// TIA Portal V20 export
// export: Created 2025-12-01T14:57:27.9326665Z, ExportSetting None, DisplayName Totally Integrated Automation Portal, DisplayVersion V20 Update 3, DisplayName TIA Portal Openness, DisplayVersion V20 Update 3, DisplayName TIA Portal Version Control Interface, DisplayVersion V20 Update 3, DisplayName STEP 7 Professional, DisplayVersion V20 Update 3, DisplayName STEP 7 Safety, DisplayVersion V20 Update 2, DisplayName WinCC Basic/Comfort/Advanced, DisplayVersion V20 Update 3, DisplayName WinCC Professional, DisplayVersion V20 Update 3, DisplayName WinCC Unified, DisplayVersion V20 Update 3
FUNCTION_BLOCK "FB602_EntradaMovil_Lateral_EnCarga_Quimarox"   // FB602, LAD
{ S7_Optimized_Access := 'FALSE' }
// stored: AutoNumber false, SetENOAutomatically false
   VAR_INPUT
      MesaAnterior : UInt;
      MesaDeCarga : UInt;
      ID_Quimarox : UInt;
      ID_Elemento : UInt;
      EnTension : Bool;
      Termico_Tx : Bool;
      Termico_Tilt : Bool;
      pHs_PosicionCarga : Bool;
      pHs_Protrusion : Bool;
      En_PosicionReposo : Bool;
      Corte_PosicionReposo : Bool;
      Corte_PosicionCarga : Bool;
      En_PosicionCarga : Bool;
      PRV_AVTF : Bool;
      PRV_DescargaActiva : Bool;
      V_FILTRO_pHsPresencia : Int;
      Pto_Ajuste_1 : Int;
      Pto_Ajuste_2 : Int;
      Pto_Ajuste_3 : Int;
      Pto_Ajuste_4 : Int;
      Pto_Ajuste_5 : Int;
      Pto_Ajuste_6 : Int;
   END_VAR
   VAR_OUTPUT
      PRV_PTF : Bool;
      PRV_FTF : Bool;
      PararElevador : Bool;
      ElevadorEnLenta : Bool;
      Avance_EntradaMovil : Bool;
      Ir_PosicionReposo : Bool;
      Ir_PosicionCarga : Bool;
   END_VAR
   VAR_IN_OUT
      ROUTING_Destino : UInt;
      ROUTING_Etiqueta : UDInt;
   END_VAR
   VAR
      TMP_EnTension { S7_SetPoint := 'True'} : "FB910_CNT_UHS";
      FILTRO_pHsPresencia { S7_SetPoint := 'True'} : "FB910_CNT_UHS";
      EstadoAsociadoEnMesa : UInt;
      Aux_PeineDeCarga : UInt;
      PresenciaEnReset : Bool;
   END_VAR
   VAR_TEMP
      TMP_PeineDeCarga : UInt;
      TMP_PeineLiberar : UInt;
      MesaQuimarox : UInt;
      VagonReservado : UInt;
      NumeroUT : UInt;
      EsMesaTL : Bool;
      FILTRO_PosicionCarga : Bool;
   END_VAR
BEGIN

NETWORK
TITLE = ERROR - Rearme
/////////////////////////////////////////////////////////////
/////////////////////////////////////////////////////////////
/////////////////////////////////////////////////////////////
// Rearne de Errores
      SET;
      A     "DB902_Estado_ZonaMesa".EstadoMesas[#MesaDeCarga].Rearme_CBx;
      O     "DB902_Estado_ZonaMesa".EstadoMesas[#MesaDeCarga].PerReset_CBx;
      R     "DB900_Estado_Mesas".EstadoVI[#MesaDeCarga].Error_Mx;
      R     "DB900_Estado_Mesas".EstadoVI[#MesaDeCarga].Err_Protusion;
      R     "DB900_Estado_Mesas".EstadoVI[#MesaDeCarga].Err_TOut_Avance_E1_E3;
      R     "DB900_Estado_Mesas".EstadoVI[#MesaDeCarga].Err_Tout_Sacar;
      R     "DB900_Estado_Mesas".EstadoVI[#MesaDeCarga].Err_Tout_Recoger;
      R     "DB900_Estado_Mesas".EstadoVI[#MesaDeCarga].Err_DatosPLC;
      R     "DB900_Estado_Mesas".EstadoVI[#MesaDeCarga].Err_Termico_E1_E3;
      R     "DB900_Estado_Mesas".EstadoVI[#MesaDeCarga].Err_Termico_E2_E4;



NETWORK
TITLE = RECEP OK DE LA ORDEN -- NO SE UTILIZA
/////////////////////////////////////////////////////////////
/////////////////////////////////////////////////////////////
/////////////////////////////////////////////////////////////
// RECEP OK DE LA ORDEN
      SET;
      AN    "DB841_Recepcion".Mesa[#MesaDeCarga].Protocolo.Ord_S00;
      AN    "DB841_Recepcion".Mesa[#MesaDeCarga].Protocolo.Ord_S01;
      AN    "DB841_Recepcion".Mesa[#MesaDeCarga].Protocolo.Ord_S02;
      AN    "DB841_Recepcion".Mesa[#MesaDeCarga].Protocolo.Ord_S03;
      NOT;
      =     "DB840_Emision".Mesa[#MesaDeCarga].Protocolo.RecepOK;



NETWORK
TITLE = HMI - Manual
/////////////////////////////////////////////////////////////
/////////////////////////////////////////////////////////////
/////////////////////////////////////////////////////////////
// Para HMI >>> Manual
      SET;
      O     "DB902_Estado_ZonaMesa".EstadoMesas[#MesaDeCarga].Manual_CBx;
      =     "DB900_Estado_Mesas".EstadoVI[#MesaDeCarga].Manual;



NETWORK
TITLE = HMI - Entradas y Salidas de la Mesa
/////////////////////////////////////////////////////////////
/////////////////////////////////////////////////////////////
/////////////////////////////////////////////////////////////
// Entradas
      SET;
      A     #pHs_PosicionCarga;
      =     "DB900_Estado_Mesas".EstadoVI[#MesaDeCarga].En_PHS_1;
      SET;
      A     #pHs_Protrusion;
      =     "DB900_Estado_Mesas".EstadoVI[#MesaDeCarga].En_pHs_Prot1;

      SET;
      A     #Termico_Tx;
      =     "DB900_Estado_Mesas".EstadoVI[#MesaDeCarga].En_Termico1;
      SET;
      A     #Termico_Tilt;
      =     "DB900_Estado_Mesas".EstadoVI[#MesaDeCarga].En_Termico2;

      SET;
      A     #En_PosicionReposo;
      =     "DB904_Estado_Maquinas".EstadoVI[#MesaDeCarga].Byte8_bit4;
      SET;
      A     #Corte_PosicionReposo;
      =     "DB904_Estado_Maquinas".EstadoVI[#MesaDeCarga].Byte7_bit6;
      SET;
      A     #Corte_PosicionCarga;
      =     "DB904_Estado_Maquinas".EstadoVI[#MesaDeCarga].Byte7_bit7;
      SET;
      A     #En_PosicionCarga;
      =     "DB904_Estado_Maquinas".EstadoVI[#MesaDeCarga].Byte8_bit5;


// Salidas
      SET;
      A     #Avance_EntradaMovil;
      =     "DB900_Estado_Mesas".EstadoVI[#MesaDeCarga].Sa_Rod_Avance;
      SET;
      A     #Ir_PosicionReposo;
      =     "DB900_Estado_Mesas".EstadoVI[#MesaDeCarga].Sa_Trans_Baj;
      SET;
      A     #Ir_PosicionCarga;
      =     "DB900_Estado_Mesas".EstadoVI[#MesaDeCarga].Sa_Trans_Sub;



NETWORK
TITLE = Comprobacion de que la MESA es de TRACKING
/////////////////////////////////////////////////////////////
/////////////////////////////////////////////////////////////
/////////////////////////////////////////////////////////////
// Comprobar si es una Mesa de Tracking o Routing
      SET;
      A     "DB850_DefinicionMesas".Mesa[#MesaDeCarga].ConfigMesa.MesaTL;
      =     #EsMesaTL;



REGION Network 6: TMP - Espera En Tension
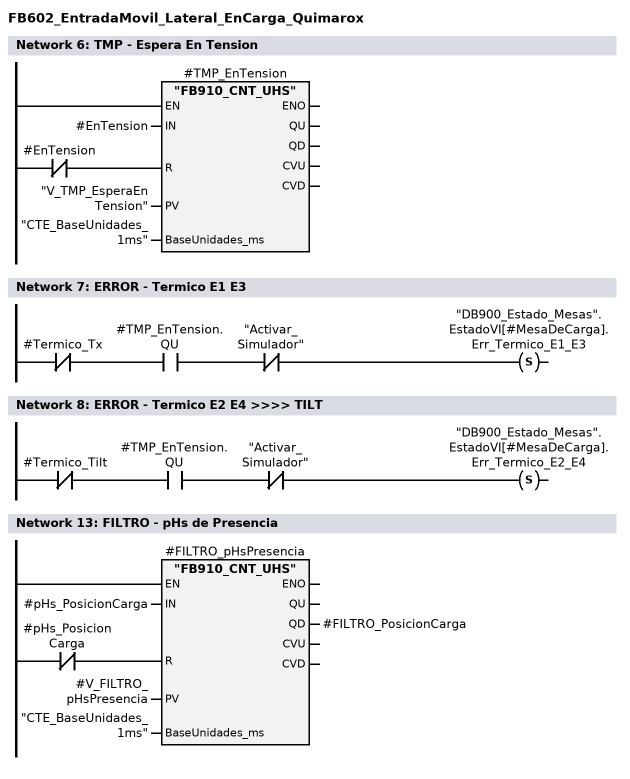
   RUNG wire#powerrail
      #TMP_EnTension(R := wire#w1, IN := #EnTension, PV := "V_TMP_EsperaEnTension", BaseUnidades_ms := "CTE_BaseUnidades_1ms", QU =>, QD =>, CVU =>, CVD =>)
   END_RUNG
   RUNG wire#powerrail
      I_Contact( #EnTension )
   END_RUNG wire#w1
   // the same network as SCL:
   #TMP_EnTension(IN := #EnTension,   // "FB910_CNT_UHS"
                  R := NOT #EnTension,
                  PV := "V_TMP_EsperaEnTension",
                  BaseUnidades_ms := "CTE_BaseUnidades_1ms");
END_REGION

REGION Network 7: ERROR - Termico E1 E3
   RUNG wire#powerrail
      I_Contact( #Termico_Tx )
      Contact( #TMP_EnTension.QU )
      I_Contact( "Activar_Simulador" )
      S_Coil( "DB900_Estado_Mesas".EstadoVI[#MesaDeCarga].Err_Termico_E1_E3 )
   END_RUNG
   // the same network as SCL:
   IF NOT #Termico_Tx AND #TMP_EnTension.QU AND NOT "Activar_Simulador" THEN
       "DB900_Estado_Mesas".EstadoVI[#MesaDeCarga].Err_Termico_E1_E3 := TRUE;
   END_IF;
END_REGION

REGION Network 8: ERROR - Termico E2 E4 >>>> TILT
   RUNG wire#powerrail
      I_Contact( #Termico_Tilt )
      Contact( #TMP_EnTension.QU )
      I_Contact( "Activar_Simulador" )
      S_Coil( "DB900_Estado_Mesas".EstadoVI[#MesaDeCarga].Err_Termico_E2_E4 )
   END_RUNG
   // the same network as SCL:
   IF NOT #Termico_Tilt AND #TMP_EnTension.QU AND NOT "Activar_Simulador" THEN
       "DB900_Estado_Mesas".EstadoVI[#MesaDeCarga].Err_Termico_E2_E4 := TRUE;
   END_IF;
END_REGION

NETWORK
TITLE = INICIALIZACION Previa
/////////////////////////////////////////////////////////////
/////////////////////////////////////////////////////////////
/////////////////////////////////////////////////////////////
      CLR;
      =     #PRV_PTF;
      =     #PRV_FTF;
      CLR;
      =     #ElevadorEnLenta;
      =     #PararElevador;
      =     #Avance_EntradaMovil;
      =     #Ir_PosicionReposo;
      =     #Ir_PosicionCarga;

      CLR;
      =     "DB900_Estado_Mesas".EstadoVI[#MesaDeCarga].Etapas_Reset;
      =     "DB900_Estado_Mesas".EstadoVI[#MesaDeCarga].Etapa_Vacia;
      =     "DB900_Estado_Mesas".EstadoVI[#MesaDeCarga].Etapa_Cargada;
      =     "DB900_Estado_Mesas".EstadoVI[#MesaDeCarga].Etapas_Carga_E1;
      =     "DB900_Estado_Mesas".EstadoVI[#MesaDeCarga].Etapas_Descarga_S0;



NETWORK
TITLE = SISTEMA - Paro Blando
/////////////////////////////////////////////////////////////
/////////////////////////////////////////////////////////////
/////////////////////////////////////////////////////////////
// - Inicializar Variables de PARO BLANDO
      CLR;
      =     "DB900_Estado_Mesas".EstadoVI[#MesaDeCarga].Paro_Blando;

/////////////////////////////////////////////////////////////
// - Existe PARO BLANDO ???
      SET;
      AN    "DB902_Estado_ZonaMesa".EstadoMesas[#MesaDeCarga].ParoBlando_CBx;
      JC    NoRealizandose_ParoBlando;

/////////////////////////////////////////////////////////////
// - Fin de PARO BLANDO
      SET;
      =     "DB900_Estado_Mesas".EstadoVI[#MesaDeCarga].Paro_Blando;


/////////////////////////////////////////////////////////////
/////////////////////////////////////////////////////////////
/////////////////////////////////////////////////////////////
// - Final Tratamiento del PARO BLANDO
NoRealizandose_ParoBlando:NOP   0;



NETWORK
TITLE = SISTEMA - Reset
/////////////////////////////////////////////////////////////
/////////////////////////////////////////////////////////////
/////////////////////////////////////////////////////////////
// -- Inicializar Variables de RESET
      SET;
      AN    "DB902_Estado_ZonaMesa".EstadoMesas[#MesaDeCarga].PerReset_CBx;
      R     "DB900_Estado_Mesas".EstadoVI[#MesaDeCarga].Fin_VI;
      R     #PresenciaEnReset;

/////////////////////////////////////////////////////////////
/////////////////////////////////////////////////////////////
/////////////////////////////////////////////////////////////
// - Existe RESET ??
      SET;
      AN    "DB902_Estado_ZonaMesa".EstadoMesas[#MesaDeCarga].PerReset_CBx;
      JC    NoRealizandose_Reset;

      L     0;  // Estado de La Mesa = 0
      T     #EstadoAsociadoEnMesa;
      SET;
      =     "DB900_Estado_Mesas".EstadoVI[#MesaDeCarga].Etapas_Reset;

/////////////////////////////////////////////////////////////
/////////////////////////////////////////////////////////////
/////////////////////////////////////////////////////////////
// - Emision de Presencia en caso de Reset
      SET;  // Presencia >>> Reset Total
      A     #FILTRO_PosicionCarga;
      AN    #PresenciaEnReset;
      A     "DB831_Mesas".Mesas[#MesaDeCarga].Memorias.M_ResetTotal;
      JC    Enviar_PresenciaEnResetTotal;

      SET;  // Presencia >>> Reset Parcial
      A     #FILTRO_PosicionCarga;
      A     "DB831_Mesas".Mesas[#MesaDeCarga].Memorias.M_ResetParcial;
      AN    #PresenciaEnReset;
      JC    Enviar_PresenciaEnResetParcial;

      JU    Final_PresenciaEnReset;

// - Presencia en Reset TOTAL >>> Enviar NUUT
Enviar_PresenciaEnResetTotal:NOP   0;
      CALL  "FC723_InsertarUT_EnMesa"
      ( MesaActual := #MesaDeCarga,
        NumeroUT   := #NumeroUT
      );
      L     132;  // Envio de Nueva UT en RESET
      T     "DB812_UTs_Control".UT[#NumeroUT].EstadoEventoAGenerar;

      SET;  // Ya esta Avisado el JdT
      S     #PresenciaEnReset;

      JU    Final_PresenciaEnReset;

// - Presencia en Reset Parcial >>> Enviar LOCA en Reset Pantalla
Enviar_PresenciaEnResetParcial:NOP   0;
      L     "DB810_ColasMesas".Colas[#MesaDeCarga].UT_PrimeraMesa;
      T     #NumeroUT;

      L     #NumeroUT;  // Comprobar que Existe UT
      L     0;
      ==I;
      JC    ErrorDatosCargada;

      L     101;  // Envio de LOCA en RESET
      T     "DB812_UTs_Control".UT[#NumeroUT].EstadoEventoAGenerar;

      SET;  // Ya esta Avisado el JdT
      S     #PresenciaEnReset;

      JU    Final_PresenciaEnReset;

// - Final de la Presencia En Reset
Final_PresenciaEnReset:NOP   0;


/////////////////////////////////////////////////////////////
/////////////////////////////////////////////////////////////
/////////////////////////////////////////////////////////////
// - Fin de RESET
      SET;  // Con Presencia de Carga >>> TOTAL
      A(;
      L     "DB810_ColasMesas".Colas[#MesaDeCarga].UT_PrimeraMesa;
      L     0;
      ==I;
      );
      A     #FILTRO_PosicionCarga;
      A     #PresenciaEnReset;
      A     "DB831_Mesas".Mesas[#MesaDeCarga].Memorias.M_ResetTotal;
      S     "DB900_Estado_Mesas".EstadoVI[#MesaDeCarga].Fin_VI;

      SET;  // Con Presencia de Carga >>> PARCIAL
      A     #FILTRO_PosicionCarga;
      A     #PresenciaEnReset;
      A     "DB831_Mesas".Mesas[#MesaDeCarga].Memorias.M_ResetParcial;
      S     "DB900_Estado_Mesas".EstadoVI[#MesaDeCarga].Fin_VI;

      SET;  // Sin Presencia de Carga
      AN    #FILTRO_PosicionCarga;
      S     "DB900_Estado_Mesas".EstadoVI[#MesaDeCarga].Fin_VI;

      BE;

/////////////////////////////////////////////////////////////
/////////////////////////////////////////////////////////////
/////////////////////////////////////////////////////////////
// - Final Tratamiento del RESET
NoRealizandose_Reset:NOP   0;



NETWORK
TITLE = >>>>>>>>>>>>>>>>>>>>>>>>>>>>>>>>>>>>>>>>>>>>>>>>>>>>>>>>>>>>>>>>>>>

REGION Network 13: FILTRO - pHs de Presencia
   RUNG wire#powerrail
      #FILTRO_pHsPresencia(R := wire#w1, IN := #pHs_PosicionCarga, PV := #V_FILTRO_pHsPresencia, BaseUnidades_ms := "CTE_BaseUnidades_1ms", QU =>, QD => #FILTRO_PosicionCarga, CVU =>, CVD =>)
   END_RUNG
   RUNG wire#powerrail
      I_Contact( #pHs_PosicionCarga )
   END_RUNG wire#w1
   // the same network as SCL:
   #FILTRO_pHsPresencia(IN := #pHs_PosicionCarga,   // "FB910_CNT_UHS"
                        R := NOT #pHs_PosicionCarga,
                        PV := #V_FILTRO_pHsPresencia,
                        BaseUnidades_ms := "CTE_BaseUnidades_1ms",
                        QD => #FILTRO_PosicionCarga);
END_REGION

NETWORK
TITLE = >>>>>>>>>>>>>>>>>>>>>>>>>>>>>>>>>>>>>>>>>>>>>>>>>>>>>>>>>>>>>>>>>>>

NETWORK
TITLE = Disrtibucion >>> Control Etapa Activa
/////////////////////////////////////////////////////////////////////////////////////
/////////////////////////////////////////////////////////////////////////////////////
/////////////////////////////////////////////////////////////////////////////////////
// listado de saltos de programa
      L     #EstadoAsociadoEnMesa;
      JL    ESTADO_PorDefecto;

      JU    ETAPA_00_EnReset;
      JU    ETAPA_01_EnReposo;

      JU    ETAPA_02_PrevioCarga_ComprobarRuta;
      JU    ETAPA_03_PrevioCarga_ReservaPeine;
      JU    ETAPA_04_PrevioCarga_Sincroniza;
      JU    ETAPA_05_PrevioCarga_MoverPosicionDeCarga;

      JU    ETAPA_06_Cargando;
      JU    ETAPA_07_FinDeCarga;
      JU    ETAPA_08_CargaDelPeine;
      JU    ETAPA_09_MoverPosicionReposo;

// --- CARGADO
      JU    ETAPA_10_Reset_MoverPosicionDeReposo;
      JU    ETAPA_11_Reset_ComprobarRuta;
      JU    ETAPA_12_Reset_ReservaPeine;
      JU    ETAPA_13_Reset_Sincroniza;
      JU    ETAPA_14_Reset_MoverPosicionDeCarga;

// --- VACIO
      JU    ETAPA_15_Reset_MoverPosicionDeReposo;

ESTADO_PorDefecto:JU    FinFuncion;







NETWORK
TITLE = ETAPA 00 >>> Etapa Reset
/////////////////////////////////////////////////////////////////////////////////////
/////////////////////////////////////////////////////////////////////////////////////
/////////////////////////////////////////////////////////////////////////////////////
ETAPA_00_EnReset:NOP   0;
      SET;
      =     "DB900_Estado_Mesas".EstadoVI[#MesaDeCarga].Etapas_Reset;


/////////////////////////////////////////////////////////////////////////////////////
// error de protusion
      SET;
      AN    #pHs_Protrusion;
      JC    ErrorProtrusion;

/////////////////////////////////////////////////////////////////////////////////////
// Tiene que estar en Marcha y Sin Error para continuar
      SET;
      AN    "DB902_Estado_ZonaMesa".EstadoMesas[#MesaDeCarga].Marcha_CBx;
      O     "DB902_Estado_ZonaMesa".EstadoMesas[#MesaDeCarga].Error_CBx;
      JC    ET00_PararElevador;


/////////////////////////////////////////////////////////////////////////////////////
/////////////////////////////////////////////////////////////////////////////////////
//  Vacio >>> No esta en Reposo
      SET;
      AN    #FILTRO_PosicionCarga;
      AN    #En_PosicionReposo;
      JC    ET00_IrEtapa_15_MoverPosicionReposo;

//  Vacio >>> Esta en Reposo
      SET;
      AN    #FILTRO_PosicionCarga;
      A     #En_PosicionReposo;
      JC    ET00_IrEtapa_01_EnReposo;


/////////////////////////////////////////////////////////////////////////////////////
/////////////////////////////////////////////////////////////////////////////////////
//  Lleno >>> No Esta en Reposo
      SET;
      A     #FILTRO_PosicionCarga;
      AN    #En_PosicionReposo;
      JC    ET00_IrEtapa_10_Reset_MoverPosicionDeReposo;

//  Lleno >>> Esta en Reposo
      SET;
      A     #FILTRO_PosicionCarga;
      A     #En_PosicionReposo;
      JC    ET00_IrEtapa_11_Reset_ComprobarRuta;

      BE;


/////////////////////////////////////////////////////////////////////////////////////
/////////////////////////////////////////////////////////////////////////////////////
/////////////////////////////////////////////////////////////////////////////////////
ET00_PararElevador:NOP   0;
      SET;
      =     #PararElevador;
      BE;


/////////////////////////////////////////////////////////////////////////////////////
/////////////////////////////////////////////////////////////////////////////////////
/////////////////////////////////////////////////////////////////////////////////////
ET00_IrEtapa_01_EnReposo:NOP   0;
      L     1;
      T     #EstadoAsociadoEnMesa;
      JU    ETAPA_01_EnReposo;

/////////////////////////////////////////////////////////////////////////////////////
ET00_IrEtapa_15_MoverPosicionReposo:NOP   0;
      L     15;
      T     #EstadoAsociadoEnMesa;
      JU    ETAPA_15_Reset_MoverPosicionDeReposo;

/////////////////////////////////////////////////////////////////////////////////////
ET00_IrEtapa_11_Reset_ComprobarRuta:NOP   0;
      L     11;
      T     #EstadoAsociadoEnMesa;
      JU    ETAPA_11_Reset_ComprobarRuta;

/////////////////////////////////////////////////////////////////////////////////////
ET00_IrEtapa_10_Reset_MoverPosicionDeReposo:NOP   0;
      L     10;
      T     #EstadoAsociadoEnMesa;
      JU    ETAPA_10_Reset_MoverPosicionDeReposo;




NETWORK
TITLE = ETAPA 01 >>> Etapa Reposo >>> Esta Vacia
/////////////////////////////////////////////////////////////////////////////////////
/////////////////////////////////////////////////////////////////////////////////////
/////////////////////////////////////////////////////////////////////////////////////
// estado reposo
ETAPA_01_EnReposo:NOP   0;
      SET;
      =     "DB900_Estado_Mesas".EstadoVI[#MesaDeCarga].Etapa_Vacia;


/////////////////////////////////////////////////////////////////////////////////////
// error de protusion
      SET;
      AN    #pHs_Protrusion;
      JC    ErrorProtrusion;

/////////////////////////////////////////////////////////////////////////////////////
/////////////////////////////////////////////////////////////////////////////////////
/////////////////////////////////////////////////////////////////////////////////////
// Si Viene un Peine >>> Reservado para el Elemento >>> LIBERAR Peine
      SET;  // --- Sin Ventana
      AN    "DB602_ElementosQuimarox".Quimarox[#ID_Quimarox].Elementos[#ID_Elemento].Hay_Carrier_en_ventana;
      JC    ET01_PorReserva_NoLiberarPeine;

      L     "DB602_ElementosQuimarox".Quimarox[#ID_Quimarox].Elementos[#ID_Elemento].Numero_carrier;
      T     #TMP_PeineLiberar;

      SET;  // --- Sin Reserva
      AN    "DB601_PeinesQuimarox".Quimarox[#ID_Quimarox].vagon[#TMP_PeineLiberar].vagon_reservado_carga;
      JC    ET01_PorReserva_NoLiberarPeine;

      SET;  // --- No es para el elemento
      L     "DB601_PeinesQuimarox".Quimarox[#ID_Quimarox].vagon[#TMP_PeineLiberar].punto_entrada_carga;
      L     #ID_Elemento;
      <>I;
      JC    ET01_PorReserva_NoLiberarPeine;

/////////////////////////////////////////////////////////////////////////////////////
      SET;  // --- Liberar Peine
      R     "DB601_PeinesQuimarox".Quimarox[#ID_Quimarox].vagon[#TMP_PeineLiberar].vagon_reservado_carga;

      L     0;
      T     "DB601_PeinesQuimarox".Quimarox[#ID_Quimarox].vagon[#TMP_PeineLiberar].punto_entrada_carga;

/////////////////////////////////////////////////////////////////////////////////////
ET01_PorReserva_NoLiberarPeine:NOP   0;


/////////////////////////////////////////////////////////////////////////////////////
// Esta poscionado Correctamente
      SET;
      AN    #PRV_AVTF;
      AN    #FILTRO_PosicionCarga;
      A     #pHs_Protrusion;
      AN    #En_PosicionReposo;
      JC    ET01_IrEtapa_09_MoverPosicionReposo;

/////////////////////////////////////////////////////////////////////////////////////
      SET;
      AN    #PRV_AVTF;
      AN    #FILTRO_PosicionCarga;
      A     #pHs_Protrusion;
      JC    FinFuncion;

/////////////////////////////////////////////////////////////////////////////////////
      SET;
      A     #PRV_AVTF;
      AN    #FILTRO_PosicionCarga;
      A     #pHs_Protrusion;
      JC    ET01_IrEtapa_02_PrevioCarga_ComprobarRuta;

      BE;


/////////////////////////////////////////////////////////////////////////////////////
ET01_IrEtapa_09_MoverPosicionReposo:NOP   0;
      L     9;
      T     #EstadoAsociadoEnMesa;
      JU    ETAPA_09_MoverPosicionReposo;

/////////////////////////////////////////////////////////////////////////////////////
ET01_IrEtapa_02_PrevioCarga_ComprobarRuta:NOP   0;
      L     2;  // tengo una caja, paso a extraer orden
      T     #EstadoAsociadoEnMesa;
      JU    ETAPA_02_PrevioCarga_ComprobarRuta;



NETWORK
TITLE = ETAPA 02 >>> Comprobar Ruta
/////////////////////////////////////////////////////////////////////////////////////
/////////////////////////////////////////////////////////////////////////////////////
/////////////////////////////////////////////////////////////////////////////////////
// Extraer Destino
ETAPA_02_PrevioCarga_ComprobarRuta:NOP   0;
      SET;
      =     "DB900_Estado_Mesas".EstadoVI[#MesaDeCarga].Etapa_Vacia;


/////////////////////////////////////////////////////////////////////////////////////
      SET;
      AN    #pHs_Protrusion;
      JC    ErrorProtrusion;

/////////////////////////////////////////////////////////////////////////////////////
/// --- Comprobacion del TIPO de MESA
      SET;
      AN    #EsMesaTL;
      JC    ET02_TRACKING_ComprobarRuta;
      JU    ET02_ROUTING_ComprobarRuta;


/////////////////////////////////////////////////////////////////////////////////////
/////////////////////////////////////////////////////////////////////////////////////
/////////////////////////////////////////////////////////////////////////////////////
/// --- Comprobacion de Ruta en una MESA de ROUTING
ET02_ROUTING_ComprobarRuta:NOP   0;
      L     #ROUTING_Destino;
      L     0;
      ==I;
      JC    FinFuncion;
      JU    ET02_FINAL_ComprobacionDeRuta;

/////////////////////////////////////////////////////////////////////////////////////
/////////////////////////////////////////////////////////////////////////////////////
/////////////////////////////////////////////////////////////////////////////////////
/// --- Comprobacion de Ruta en una MESA de TRACKING
ET02_TRACKING_ComprobarRuta:NOP   0;
      L     "DB810_ColasMesas".Colas[#MesaAnterior].UT_PrimeraMesa;
      T     #NumeroUT;

      SET;
      L     #NumeroUT;  // Debe existir UT
      L     0;
      ==I;
      JC    FinFuncion;

// si la mesa actual es la de destino, es que aun no tiene ruta, y tenemos que esperar
      SET;
      L     "DB812_UTs_Control".UT[#NumeroUT].MesaActual;
      L     "DB812_UTs_Control".UT[#NumeroUT].MesaDestino;
      ==I;
      JC    FinFuncion;

      SET;
      L     0;
      L     "DB812_UTs_Control".UT[#NumeroUT].MesaDestino;
      ==I;
      JC    FinFuncion;

      JU    ET02_FINAL_ComprobacionDeRuta;

/////////////////////////////////////////////////////////////////////////////////////
/////////////////////////////////////////////////////////////////////////////////////
/////////////////////////////////////////////////////////////////////////////////////
/// --- Final de la Comprobacion de Ruta
//      si tenemos destino, pasamos a reservar peine de carga
ET02_FINAL_ComprobacionDeRuta:NOP   0;
      L     3;
      T     #EstadoAsociadoEnMesa;
      JU    ETAPA_03_PrevioCarga_ReservaPeine;  // si ya hemos extraido la orden, pasamos a extraer el destino



NETWORK
TITLE = ETAPA 03 >>> Reserva Peine
/////////////////////////////////////////////////////////////////////////////////////
/////////////////////////////////////////////////////////////////////////////////////
/////////////////////////////////////////////////////////////////////////////////////
// reserva de peine
ETAPA_03_PrevioCarga_ReservaPeine:NOP   0;
      SET;
      =     "DB900_Estado_Mesas".EstadoVI[#MesaDeCarga].Etapa_Vacia;


/////////////////////////////////////////////////////////////////////////////////////
// revisamos error de protusion
      SET;
      AN    #pHs_Protrusion;
      JC    ErrorProtrusion;

/////////////////////////////////////////////////////////////////////////////////////
// rearme del error si ha desaparecido la caja   OJO!!!!!!!CAMBIADO
      SET;
      AN    #PRV_AVTF;
      AN    #FILTRO_PosicionCarga;
      A     #pHs_Protrusion;
      A     "DB902_Estado_ZonaMesa".EstadoMesas[#MesaDeCarga].Rearme_CBx;
      JC    ET03_IrEtapa_01_EnReposo;


/////////////////////////////////////////////////////////////////////////////////////
/////////////////////////////////////////////////////////////////////////////////////
/////////////////////////////////////////////////////////////////////////////////////
// reserva de peine >>> Mesa Movil Lateral (2)
      CALL  "FC602_ReservaPeine"
      ( ID_Quimarox          := #ID_Quimarox,
        ID_ElementoPeticion  := #ID_Elemento,
        TipoDeElemento       := 2,
        NumeroPeineReservado := #VagonReservado
      );

      SET;
      L     #VagonReservado;
      L     0;
      ==I;
      JC    FinFuncion;

/////////////////////////////////////////////////////////////////////////////////////
/////////////////////////////////////////////////////////////////////////////////////
/////////////////////////////////////////////////////////////////////////////////////
      L     #VagonReservado;  // recogemos la peticion
      T     #Aux_PeineDeCarga;

      L     4;
      T     #EstadoAsociadoEnMesa;
      JU    ETAPA_04_PrevioCarga_Sincroniza;


/////////////////////////////////////////////////////////////////////////////////////
ET03_IrEtapa_01_EnReposo:NOP   0;
      L     1;
      T     #EstadoAsociadoEnMesa;
      JU    ETAPA_01_EnReposo;



NETWORK
TITLE = ETAPA 04 >>> Sincronizacion
/////////////////////////////////////////////////////////////////////////////////////
/////////////////////////////////////////////////////////////////////////////////////
/////////////////////////////////////////////////////////////////////////////////////
// a la espera de la sincronización con el peine reservado para nosotros
ETAPA_04_PrevioCarga_Sincroniza:NOP   0;
      SET;
      =     "DB900_Estado_Mesas".EstadoVI[#MesaDeCarga].Etapas_Carga_E1;


/////////////////////////////////////////////////////////////////////////////////////
// revisamos error de protusion
      SET;
      AN    #pHs_Protrusion;
      JC    ErrorProtrusion;

/////////////////////////////////////////////////////////////////////////////////////
// ahora que ya estamos los datos de nuestro elemento comprobamos lo siguiente
// que tenemos delante el carrier que tenemos reservado para la carga
// que el carrier reservado para la carga está en ventana
      SET;
      A     "DB602_ElementosQuimarox".Quimarox[#ID_Quimarox].Elementos[#ID_Elemento].Hay_Carrier_en_ventana;
      A(;
      L     "DB602_ElementosQuimarox".Quimarox[#ID_Quimarox].Elementos[#ID_Elemento].Numero_carrier;  //#datos_elemento.Numero_carrier
      L     #Aux_PeineDeCarga;
      ==I;
      );
      JC    ET04_IrEtapa_05_MoverPosicionDeCarga;

      BE;


/////////////////////////////////////////////////////////////////////////////////////
ET04_IrEtapa_05_MoverPosicionDeCarga:NOP   0;
      L     5;  // saltamos al inicio de posicionamiento para carga
      T     #EstadoAsociadoEnMesa;
      JU    ETAPA_05_PrevioCarga_MoverPosicionDeCarga;



NETWORK
TITLE = ETAPA 05 >>> Mover Posicion de Carga >>> INICIO del Movimiento
/////////////////////////////////////////////////////////////////////////////////////
/////////////////////////////////////////////////////////////////////////////////////
/////////////////////////////////////////////////////////////////////////////////////
ETAPA_05_PrevioCarga_MoverPosicionDeCarga:NOP   0;
      SET;
      =     "DB900_Estado_Mesas".EstadoVI[#MesaDeCarga].Etapas_Carga_E1;


/////////////////////////////////////////////////////////////////////////////////////
      SET;
      A     #En_PosicionCarga;
      JC    ET05_IrEtapa_06_Cargando;

      SET;
      =     #Ir_PosicionCarga;
      CLR;
      =     #Ir_PosicionReposo;


/////////////////////////////////////////////////////////////////////////////////////
/////////////////////////////////////////////////////////////////////////////////////
// como estamos metiendo el transportador, tenemos que vigilar que no tarda demasiado en entrar
      L     "DB602_ElementosQuimarox".Quimarox[#ID_Quimarox].Elementos[#ID_Elemento].Avance_carrier;
      L     #Pto_Ajuste_1;
      <=I;
      JC    ET05_VelocidadNormal;

      SET;
      =     #ElevadorEnLenta;

/////////////////////////////////////////////////////////////////////////////////////
      L     "DB602_ElementosQuimarox".Quimarox[#ID_Quimarox].Elementos[#ID_Elemento].Avance_carrier;
      L     #Pto_Ajuste_2;
      >=I;
      JC    ErrorMoverPosicionCarga;  // error de movimiento al sacar el transportador

      BE;


/////////////////////////////////////////////////////////////////////////////////////
ET05_VelocidadNormal:CLR;
      =     #ElevadorEnLenta;
      BE;

/////////////////////////////////////////////////////////////////////////////////////
ET05_IrEtapa_06_Cargando:NOP   0;
      CLR;
      =     #Ir_PosicionCarga;

      L     6;
      T     #EstadoAsociadoEnMesa;
      JU    ETAPA_06_Cargando;



NETWORK
TITLE = ETAPA 06 >>> Cargando >>> Entrada
/////////////////////////////////////////////////////////////////////////////////////
/////////////////////////////////////////////////////////////////////////////////////
/////////////////////////////////////////////////////////////////////////////////////
ETAPA_06_Cargando:NOP   0;
      SET;
      =     "DB900_Estado_Mesas".EstadoVI[#MesaDeCarga].Etapas_Carga_E1;


/////////////////////////////////////////////////////////////////////////////////////
      SET;
      =     #PRV_PTF;
      =     #Avance_EntradaMovil;

/////////////////////////////////////////////////////////////////////////////////////
// hemos cargado correctamente y generamos los datos para el peine
      SET;
      A     #FILTRO_PosicionCarga;
      A     #PRV_AVTF;
      A     #pHs_Protrusion;
      JC    ET06_IrEtapa_07_FinCargaDelPeine;

/////////////////////////////////////////////////////////////////////////////////////
// aqui tenemos que vigilar que nos se nos está cerrado la ventana intentando cargar
// primero comprobamos que no tenemos ya la ventana cerrada, porque sino tenemos que parar el elevador
      SET;
      AN    "DB602_ElementosQuimarox".Quimarox[#ID_Quimarox].Elementos[#ID_Elemento].Hay_Carrier_en_ventana;
      A(;
      ON    #pHs_Protrusion;
      O     #FILTRO_PosicionCarga;
      );
      JC    ErrorEnCarga;

/////////////////////////////////////////////////////////////////////////////////////
      SET;
      AN    "DB602_ElementosQuimarox".Quimarox[#ID_Quimarox].Elementos[#ID_Elemento].Hay_Carrier_en_ventana;
      AN    #FILTRO_PosicionCarga;
      A     #pHs_Protrusion;
      AN    #PRV_AVTF;
      JC    ET06_PasadoVagon_SinCargar;

/////////////////////////////////////////////////////////////////////////////////////
// Deberia Haber Cargado en este punto
      SET;
      A     "DB602_ElementosQuimarox".Quimarox[#ID_Quimarox].Elementos[#ID_Elemento].Hay_Carrier_en_ventana;
      A(;
      L     "DB602_ElementosQuimarox".Quimarox[#ID_Quimarox].Elementos[#ID_Elemento].Avance_carrier;
      L     #Pto_Ajuste_4;
      >=I;
      );
      AN    #pHs_Protrusion;
      JC    ErrorProtrusion;

/////////////////////////////////////////////////////////////////////////////////////
// si seguimos teniendo el carrier en ventana, comprobamos cuanta ventana tenemos.
// llegados a un punto, pasaremos a lenta
      SET;
      A(;
      L     "DB602_ElementosQuimarox".Quimarox[#ID_Quimarox].Elementos[#ID_Elemento].Avance_carrier;
      L     #Pto_Ajuste_3;
      >=I;
      );
      JC    ET06_ElevadorLenta;

/////////////////////////////////////////////////////////////////////////////////////
      BE;


/////////////////////////////////////////////////////////////////////////////////////
ET06_ElevadorLenta:SET;
      =     #ElevadorEnLenta;
      BE;


/////////////////////////////////////////////////////////////////////////////////////
ET06_PasadoVagon_SinCargar:NOP   0;
      CLR;
      =     #ElevadorEnLenta;
      =     #PRV_PTF;
      =     #Avance_EntradaMovil;

      CLR;
      =     "DB601_PeinesQuimarox".Quimarox[#ID_Quimarox].vagon[#Aux_PeineDeCarga].vagon_reservado_carga;  //#datos_peine_tmp.vagon_reservado_carga
      L     0;
      T     "DB601_PeinesQuimarox".Quimarox[#ID_Quimarox].vagon[#Aux_PeineDeCarga].punto_entrada_carga;
      T     #Aux_PeineDeCarga;

      L     9;
      T     #EstadoAsociadoEnMesa;
      JU    ETAPA_09_MoverPosicionReposo;


/////////////////////////////////////////////////////////////////////////////////////
ET06_IrEtapa_07_FinCargaDelPeine:NOP   0;
      L     7;
      T     #EstadoAsociadoEnMesa;

/////////////////////////////////////////////////////////////////////////////////////
// - Comprobacion del TIPO de MESA
      SET;
      A     #EsMesaTL;
      JC    ETAPA_07_FinDeCarga;

// - Traer la UT de la Mesa Anterior
      L     "DB810_ColasMesas".Colas[#MesaAnterior].UT_PrimeraMesa;
      T     #NumeroUT;

      SET;  // No existe UT >>> Error de Datos
      L     #NumeroUT;
      L     0;
      ==I;
      JC    ErrorDatosCargada;

      CALL  "FC724_CambiarUT_DeMesa"
      ( NumeroUT    := #NumeroUT,
        NuevaMesa   := #MesaDeCarga,
        AlPrincipio := "DB850_DefinicionMesas".Mesa[#MesaDeCarga].ConfigMesa.MeterAlPrincipio
      );  // Cambia la UT a la Nueva Mesa

      L     0;  // Es de Ordenes Especiales - Resetear
      T     "DB812_UTs_Control".UT[#NumeroUT].EstadoRecepcionUT;
      T     "DB812_UTs_Control".UT[#NumeroUT].EstadoEventoRecibido;
      T     "DB812_UTs_Control".UT[#NumeroUT].EstadoEmisionUT;
      L     100;  // Emitir evento LOCA
      T     "DB812_UTs_Control".UT[#NumeroUT].EstadoEventoAGenerar;

      JU    ETAPA_07_FinDeCarga;



NETWORK
TITLE = ETAPA 07 >>> Fin de la Carga >>> Cargada
/////////////////////////////////////////////////////////////////////////////////////
/////////////////////////////////////////////////////////////////////////////////////
/////////////////////////////////////////////////////////////////////////////////////
ETAPA_07_FinDeCarga:NOP   0;
      SET;
      =     "DB900_Estado_Mesas".EstadoVI[#MesaDeCarga].Etapas_Carga_E1;


/////////////////////////////////////////////////////////////////////////////////////
      SET;
      =     #PRV_FTF;
      CLR;
      =     #PRV_PTF;
      =     #Avance_EntradaMovil;

/////////////////////////////////////////////////////////////////////////////////////
// Error de Protrusion
      SET;
      AN    #pHs_Protrusion;
      JC    ErrorProtrusion;

/////////////////////////////////////////////////////////////////////////////////////
// Cargado Correctamente
      SET;
      A     #FILTRO_PosicionCarga;
      A     #pHs_Protrusion;
      AN    #PRV_AVTF;
      AN    #PRV_DescargaActiva;
      JC    ET06_IrEtapa_08_CargaDelPeine;

      BE;


/////////////////////////////////////////////////////////////////////////////////////
/////////////////////////////////////////////////////////////////////////////////////
/////////////////////////////////////////////////////////////////////////////////////
ET06_IrEtapa_08_CargaDelPeine:NOP   0;
      L     8;
      T     #EstadoAsociadoEnMesa;
      JU    ETAPA_08_CargaDelPeine;



NETWORK
TITLE = ETAPA 08 >>> Fin de Carga del Peine >>> Paso de Datos al VAGON
/////////////////////////////////////////////////////////////////////////////////////
/////////////////////////////////////////////////////////////////////////////////////
/////////////////////////////////////////////////////////////////////////////////////
ETAPA_08_CargaDelPeine:NOP   0;
      SET;
      =     "DB900_Estado_Mesas".EstadoVI[#MesaDeCarga].Etapas_Descarga_S0;


/////////////////////////////////////////////////////////////////////////////////////
      CLR;
      =     #PRV_PTF;
      =     #PRV_FTF;
      =     #Avance_EntradaMovil;
      =     #ElevadorEnLenta;

      L     "DB602_ElementosQuimarox".Quimarox[#ID_Quimarox].Elementos[#ID_Elemento].Numero_carrier;
      T     #TMP_PeineDeCarga;  // Peine que esta pasando por el Elemento


/////////////////////////////////////////////////////////////////////////////////////
// Error de Protrusion
      SET;
      AN    #pHs_Protrusion;
      JC    ErrorProtrusion;

/////////////////////////////////////////////////////////////////////////////////////
// Cargado Correctamente en el PEINE
      SET;
      AN    #FILTRO_PosicionCarga;
      A     #pHs_Protrusion;
      JC    FINALIZADO_CargaDelPeine;

      BE;


/////////////////////////////////////////////////////////////////////////////////////
/////////////////////////////////////////////////////////////////////////////////////
/////////////////////////////////////////////////////////////////////////////////////
// cargamos los datos de la UT al peine   >>>>> DEPENDIENDO DE TIPO DE DATOS
FINALIZADO_CargaDelPeine:NOP   0;

// Numero de Peine que lo ha recogido  ?????? CUIDADO
      L     #TMP_PeineDeCarga;
      T     #Aux_PeineDeCarga;

// Tipo de Mesa ROUTING o TRACKING
      SET;
      =     "DB601_PeinesQuimarox".Quimarox[#ID_Quimarox].vagon[#Aux_PeineDeCarga].Carrier_Cargado;

      SET;
      AN    #EsMesaTL;
      JC    TRACKING_PasoDeDatos;
      JU    ROUTING_PasoDeDatos;

/////////////////////////////////////////////////////////////////////////////////////
// --- DATOS DE ROUTING
ROUTING_PasoDeDatos:NOP   0;
      L     0;
      T     "DB601_PeinesQuimarox".Quimarox[#ID_Quimarox].vagon[#Aux_PeineDeCarga].DatosCarga.Mckey;
      L     #MesaDeCarga;
      T     "DB601_PeinesQuimarox".Quimarox[#ID_Quimarox].vagon[#Aux_PeineDeCarga].DatosCarga.MesaOrigen;
      L     #ROUTING_Destino;
      T     "DB601_PeinesQuimarox".Quimarox[#ID_Quimarox].vagon[#Aux_PeineDeCarga].DatosCarga.MesaDestino;
      T     "DB601_PeinesQuimarox".Quimarox[#ID_Quimarox].vagon[#Aux_PeineDeCarga].Destino_principal;

      L     #ROUTING_Etiqueta;
      T     "DB601_PeinesQuimarox".Quimarox[#ID_Quimarox].vagon[#Aux_PeineDeCarga].DatosCarga.EtiquetaRouter;

      L     "CTE_Evento_QCAR";
      T     "DB601_PeinesQuimarox".Quimarox[#ID_Quimarox].vagon[#Aux_PeineDeCarga].EventoAGenerar;

      L     0;
      T     #ROUTING_Destino;
      T     #ROUTING_Etiqueta;

      JU    FINAL_PasoDeDatos;

/////////////////////////////////////////////////////////////////////////////////////
// --- DATOS DE TRACKING
TRACKING_PasoDeDatos:NOP   0;
      L     "DB810_ColasMesas".Colas[#MesaDeCarga].UT_PrimeraMesa;
      T     #NumeroUT;

      L     "DB812_UTs_Control".UT[#NumeroUT].Mckey;
      T     "DB601_PeinesQuimarox".Quimarox[#ID_Quimarox].vagon[#Aux_PeineDeCarga].DatosCarga.Mckey;
      L     "DB812_UTs_Control".UT[#NumeroUT].MesaActual;
      T     "DB601_PeinesQuimarox".Quimarox[#ID_Quimarox].vagon[#Aux_PeineDeCarga].DatosCarga.MesaOrigen;
      L     "DB812_UTs_Control".UT[#NumeroUT].MesaDestino;
      T     "DB601_PeinesQuimarox".Quimarox[#ID_Quimarox].vagon[#Aux_PeineDeCarga].DatosCarga.MesaDestino;
      T     "DB601_PeinesQuimarox".Quimarox[#ID_Quimarox].vagon[#Aux_PeineDeCarga].Destino_principal;

      L     "DB814_UTs_Etiqueta".UT[#NumeroUT].EtiquetaRouter;
      T     "DB601_PeinesQuimarox".Quimarox[#ID_Quimarox].vagon[#Aux_PeineDeCarga].DatosCarga.EtiquetaRouter;

      L     "CTE_Evento_QCAR";
      T     "DB601_PeinesQuimarox".Quimarox[#ID_Quimarox].vagon[#Aux_PeineDeCarga].EventoAGenerar;
      L     131;
      T     "DB812_UTs_Control".UT[#NumeroUT].EstadoEventoAGenerar;

// Borrar UT Sin Avisar al JDT >>>> OJO
      CALL  "FC722_EliminarUT_DeMesa"
      ( NumeroUT := #NumeroUT
      );


/////////////////////////////////////////////////////////////////////////////////////
/////////////////////////////////////////////////////////////////////////////////////
/////////////////////////////////////////////////////////////////////////////////////
FINAL_PasoDeDatos:NOP   0;
      CLR;
      =     "DB601_PeinesQuimarox".Quimarox[#ID_Quimarox].vagon[#Aux_PeineDeCarga].vagon_reservado_carga;  //#datos_peine_tmp.vagon_reservado_carga

      L     0;
      T     "DB601_PeinesQuimarox".Quimarox[#ID_Quimarox].vagon[#Aux_PeineDeCarga].punto_entrada_carga;
      T     #Aux_PeineDeCarga;

// pasamos a la etapa de volver a posicion de reposo
      L     9;
      T     #EstadoAsociadoEnMesa;
      JU    ETAPA_09_MoverPosicionReposo;



NETWORK
TITLE = ETAPA 09 >>> Mover Posicion de Reposo >>> FINAL del Movimiento
/////////////////////////////////////////////////////////////////////////////////////
/////////////////////////////////////////////////////////////////////////////////////
/////////////////////////////////////////////////////////////////////////////////////
ETAPA_09_MoverPosicionReposo:NOP   0;
      SET;
      =     "DB900_Estado_Mesas".EstadoVI[#MesaDeCarga].Etapa_Vacia;


/////////////////////////////////////////////////////////////////////////////////////
      SET;
      A     #En_PosicionReposo;
      JC    ET09_IrEtapa_01_Vacia;

      SET;
      =     #Ir_PosicionReposo;
      CLR;
      =     #Ir_PosicionCarga;


/////////////////////////////////////////////////////////////////////////////////////
/////////////////////////////////////////////////////////////////////////////////////
/////////////////////////////////////////////////////////////////////////////////////
      SET;
      L     "DB602_ElementosQuimarox".Quimarox[#ID_Quimarox].Elementos[#ID_Elemento].Avance_carrier;
      L     #Pto_Ajuste_5;
      <=I;
      JC    ET09_VelocidadNormal;

      SET;
      =     #ElevadorEnLenta;

/////////////////////////////////////////////////////////////////////////////////////
// error de movimiento al meter el transportador
      SET;
      L     "DB602_ElementosQuimarox".Quimarox[#ID_Quimarox].Elementos[#ID_Elemento].Avance_carrier;
      L     #Pto_Ajuste_6;
      >=I;
      JC    ErrorMoverPosicionReposo;

/////////////////////////////////////////////////////////////////////////////////////
// Si ya no Ventana
      SET;
      AN    "DB602_ElementosQuimarox".Quimarox[#ID_Quimarox].Elementos[#ID_Elemento].Hay_Carrier_en_ventana;
      JC    ErrorMoverPosicionReposo;

      BE;


/////////////////////////////////////////////////////////////////////////////////////
ET09_VelocidadNormal:NOP   0;
      CLR;
      =     #ElevadorEnLenta;
      BE;

/////////////////////////////////////////////////////////////////////////////////////
ET09_IrEtapa_01_Vacia:NOP   0;
      CLR;
      =     #Ir_PosicionReposo;
      =     #Ir_PosicionCarga;
      =     #ElevadorEnLenta;

      L     1;
      T     #EstadoAsociadoEnMesa;
      BE;



NETWORK
TITLE = >>>>>>>>>>>>>>>>>>>>>>>>>>>>>>>>>>>>>>>>>>>>>>>>>>>>>>>>>>>>>>>>>>>

NETWORK
TITLE = ETAPA 10 >>> RESET CARGADO >>> Mover Posicion de Reposo
/////////////////////////////////////////////////////////////////////////////////////
/////////////////////////////////////////////////////////////////////////////////////
/////////////////////////////////////////////////////////////////////////////////////
ETAPA_10_Reset_MoverPosicionDeReposo:NOP   0;
      SET;
      =     "DB900_Estado_Mesas".EstadoVI[#MesaDeCarga].Etapas_Reset;


/////////////////////////////////////////////////////////////////////////////////////
      SET;
      A     #En_PosicionReposo;
      JC    ET10_IrEtapa_11_Reset_ComprobarRuta;


/////////////////////////////////////////////////////////////////////////////////////
      SET;
      =     #Ir_PosicionReposo;
      =     #PararElevador;
      CLR;
      =     #Ir_PosicionCarga;

/////////////////////////////////////////////////////////////////////////////////////
      SET;
      AN    #pHs_Protrusion;
      JC    ErrorProtrusion;

      BE;


/////////////////////////////////////////////////////////////////////////////////////
/////////////////////////////////////////////////////////////////////////////////////
/////////////////////////////////////////////////////////////////////////////////////
ET10_IrEtapa_11_Reset_ComprobarRuta:NOP   0;
      CLR;
      =     #Ir_PosicionReposo;
      =     #Ir_PosicionCarga;

      L     11;
      T     #EstadoAsociadoEnMesa;
      JU    ETAPA_11_Reset_ComprobarRuta;



NETWORK
TITLE = ETAPA 11 >>> RESET CARGADO >>> Comprobar Ruta
/////////////////////////////////////////////////////////////////////////////////////
/////////////////////////////////////////////////////////////////////////////////////
// Extraer Destino
ETAPA_11_Reset_ComprobarRuta:NOP   0;
      SET;
      =     "DB900_Estado_Mesas".EstadoVI[#MesaDeCarga].Etapas_Reset;


/////////////////////////////////////////////////////////////////////////////////////
      SET;
      =     #PararElevador;
      CLR;
      =     #Ir_PosicionCarga;
      =     #Ir_PosicionReposo;


/////////////////////////////////////////////////////////////////////////////////////
      SET;
      AN    #pHs_Protrusion;
      JC    ErrorProtrusion;


/////////////////////////////////////////////////////////////////////////////////////
/// --- Comprobacion del TIPO de MESA
      SET;
      AN    #EsMesaTL;
      JC    ET11_TRACKING_ComprobarRuta;
      JU    ET11_ROUTING_ComprobarRuta;


/////////////////////////////////////////////////////////////////////////////////////
/////////////////////////////////////////////////////////////////////////////////////
/////////////////////////////////////////////////////////////////////////////////////
/// --- Comprobacion de Ruta en una MESA de ROUTING
ET11_ROUTING_ComprobarRuta:NOP   0;
      L     #ROUTING_Destino;
      L     0;
      ==I;
      JC    ErrorDatosCargada;
      JU    ET11_FINAL_ComprobacionDeRuta;

/////////////////////////////////////////////////////////////////////////////////////
/////////////////////////////////////////////////////////////////////////////////////
/////////////////////////////////////////////////////////////////////////////////////
/// --- Comprobacion de Ruta en una MESA de TRACKING
ET11_TRACKING_ComprobarRuta:NOP   0;
      L     "DB810_ColasMesas".Colas[#MesaDeCarga].UT_PrimeraMesa;
      T     #NumeroUT;

      SET;
      L     #NumeroUT;  // Debe existir UT
      L     0;
      ==I;
      JC    ErrorDatosCargada;

// si la mesa actual es la de destino, es que aun no tiene ruta, y tenemos que esperar
      SET;
      L     "DB812_UTs_Control".UT[#NumeroUT].MesaActual;
      L     "DB812_UTs_Control".UT[#NumeroUT].MesaDestino;
      ==I;
      JC    FinFuncion;

      SET;
      L     0;
      L     "DB812_UTs_Control".UT[#NumeroUT].MesaDestino;
      ==I;
      JC    FinFuncion;

      JU    ET11_FINAL_ComprobacionDeRuta;

/////////////////////////////////////////////////////////////////////////////////////
/////////////////////////////////////////////////////////////////////////////////////
/////////////////////////////////////////////////////////////////////////////////////
/// --- Final de la Comprobacion de Ruta
//      si tenemos destino, pasamos a reservar peine de carga
ET11_FINAL_ComprobacionDeRuta:NOP   0;
      L     12;
      T     #EstadoAsociadoEnMesa;
      JU    ETAPA_12_Reset_ReservaPeine;  // si ya hemos extraido la orden, pasamos a extraer el destino




NETWORK
TITLE = ETAPA 12 >>> RESET CARGADO >>> Reserva Peine
/////////////////////////////////////////////////////////////////////////////////////
/////////////////////////////////////////////////////////////////////////////////////
/////////////////////////////////////////////////////////////////////////////////////
// reserva de peine
ETAPA_12_Reset_ReservaPeine:NOP   0;
      SET;
      =     "DB900_Estado_Mesas".EstadoVI[#MesaDeCarga].Etapas_Reset;


/////////////////////////////////////////////////////////////////////////////////////
// revisamos error de protusion
      SET;
      AN    #pHs_Protrusion;
      JC    ErrorProtrusion;


/////////////////////////////////////////////////////////////////////////////////////
/////////////////////////////////////////////////////////////////////////////////////
/////////////////////////////////////////////////////////////////////////////////////
// reserva de peine >>> Mesa Movil Lateral (2)
      CALL  "FC602_ReservaPeine"
      ( ID_Quimarox          := #ID_Quimarox,
        ID_ElementoPeticion  := #ID_Elemento,
        TipoDeElemento       := 2,
        NumeroPeineReservado := #VagonReservado
      );

      SET;
      L     #VagonReservado;
      L     0;
      ==I;
      JC    FinFuncion;

/////////////////////////////////////////////////////////////////////////////////////
/////////////////////////////////////////////////////////////////////////////////////
/////////////////////////////////////////////////////////////////////////////////////
      L     #VagonReservado;  // recogemos la peticion
      T     #Aux_PeineDeCarga;

      JU    ET12_IrEtapa_13_Reset_Sincroniza;


/////////////////////////////////////////////////////////////////////////////////////
ET12_IrEtapa_13_Reset_Sincroniza:NOP   0;
      L     13;
      T     #EstadoAsociadoEnMesa;
      JU    ETAPA_13_Reset_Sincroniza;




NETWORK
TITLE = ETAPA 13 >>> RESET CARGADO >>> Sincronizar
/////////////////////////////////////////////////////////////////////////////////////
/////////////////////////////////////////////////////////////////////////////////////
/////////////////////////////////////////////////////////////////////////////////////
// a la espera de la sincronización con el peine reservado para nosotros
ETAPA_13_Reset_Sincroniza:NOP   0;
      SET;
      =     "DB900_Estado_Mesas".EstadoVI[#MesaDeCarga].Etapas_Reset;


/////////////////////////////////////////////////////////////////////////////////////
// revisamos error de protusion
      SET;
      AN    #pHs_Protrusion;
      JC    ErrorProtrusion;

/////////////////////////////////////////////////////////////////////////////////////
// ahora que ya estamos los datos de nuestro elemento comprobamos lo siguiente
// que tenemos delante el carrier que tenemos reservado para la carga
// que el carrier reservado para la carga está en ventana
      SET;
      A     "DB602_ElementosQuimarox".Quimarox[#ID_Quimarox].Elementos[#ID_Elemento].Hay_Carrier_en_ventana;
      A(;
      L     "DB602_ElementosQuimarox".Quimarox[#ID_Quimarox].Elementos[#ID_Elemento].Numero_carrier;  //#datos_elemento.Numero_carrier
      L     #Aux_PeineDeCarga;
      ==I;
      );
      JC    ET13_IrEtapa_14_MoverPosicionDeCarga;

      BE;


/////////////////////////////////////////////////////////////////////////////////////
ET13_IrEtapa_14_MoverPosicionDeCarga:NOP   0;
      L     14;
      T     #EstadoAsociadoEnMesa;
      JU    ETAPA_14_Reset_MoverPosicionDeCarga;



NETWORK
TITLE = ETAPA 14 >>> RESET CARGADO >>> Mover Posicion de Carga
/////////////////////////////////////////////////////////////////////////////////////
/////////////////////////////////////////////////////////////////////////////////////
/////////////////////////////////////////////////////////////////////////////////////
ETAPA_14_Reset_MoverPosicionDeCarga:NOP   0;
      SET;
      =     "DB900_Estado_Mesas".EstadoVI[#MesaDeCarga].Etapas_Descarga_S0;


/////////////////////////////////////////////////////////////////////////////////////
      SET;
      A     #En_PosicionCarga;
      JC    ET14_IrEtapa_08_CargaDelPeine;

      SET;
      =     #Ir_PosicionCarga;
      CLR;
      =     #Ir_PosicionReposo;


/////////////////////////////////////////////////////////////////////////////////////
/////////////////////////////////////////////////////////////////////////////////////
// como estamos metiendo el transportador, tenemos que vigilar que no tarda demasiado en entrar
      L     "DB602_ElementosQuimarox".Quimarox[#ID_Quimarox].Elementos[#ID_Elemento].Avance_carrier;
      L     #Pto_Ajuste_1;
      <=I;
      JC    ET14_VelocidadNormal;

      SET;
      =     #ElevadorEnLenta;

/////////////////////////////////////////////////////////////////////////////////////
      L     "DB602_ElementosQuimarox".Quimarox[#ID_Quimarox].Elementos[#ID_Elemento].Avance_carrier;
      L     #Pto_Ajuste_2;
      >=I;
      JC    ErrorMoverPosicionCarga;  // error de movimiento al sacar el transportador

      BE;


/////////////////////////////////////////////////////////////////////////////////////
ET14_VelocidadNormal:CLR;
      =     #ElevadorEnLenta;
      BE;

/////////////////////////////////////////////////////////////////////////////////////
ET14_IrEtapa_08_CargaDelPeine:NOP   0;
      CLR;
      =     #Ir_PosicionCarga;

      L     8;
      T     #EstadoAsociadoEnMesa;
      JU    ETAPA_08_CargaDelPeine;



NETWORK
TITLE = ETAPA 15 >>> RESET VACIO >>> Mover Posicion de Reposo
/////////////////////////////////////////////////////////////////////////////////////
/////////////////////////////////////////////////////////////////////////////////////
/////////////////////////////////////////////////////////////////////////////////////
ETAPA_15_Reset_MoverPosicionDeReposo:NOP   0;
      SET;
      =     "DB900_Estado_Mesas".EstadoVI[#MesaDeCarga].Etapas_Reset;


/////////////////////////////////////////////////////////////////////////////////////
      SET;
      A     #En_PosicionReposo;
      JC    ET15_IrEtapa_1_Reset_EnReposo;


/////////////////////////////////////////////////////////////////////////////////////
      SET;
      =     #Ir_PosicionReposo;
      =     #PararElevador;
      CLR;
      =     #Ir_PosicionCarga;

/////////////////////////////////////////////////////////////////////////////////////
      SET;
      AN    #pHs_Protrusion;
      JC    ErrorProtrusion;

      BE;


/////////////////////////////////////////////////////////////////////////////////////
/////////////////////////////////////////////////////////////////////////////////////
/////////////////////////////////////////////////////////////////////////////////////
ET15_IrEtapa_1_Reset_EnReposo:NOP   0;
      CLR;
      =     #Ir_PosicionReposo;
      =     #Ir_PosicionCarga;

      L     1;
      T     #EstadoAsociadoEnMesa;
      JU    ETAPA_01_EnReposo;


NETWORK
TITLE = >>>>>>>>>>>>>>>>>>>>>>>>>>>>>>>>>>>>>>>>>>>>>>>>>>>>>>>>>>>>>>>>>>>

NETWORK
TITLE = ERRRORES DE LA MESA >>> Activacion
/////////////////////////////////////////////////////////////////////////////////////
/////////////////////////////////////////////////////////////////////////////////////
/////////////////////////////////////////////////////////////////////////////////////
ErrorProtrusion:NOP   0;
      SET;
      =     "DB900_Estado_Mesas".EstadoVI[#MesaDeCarga].Error_Mx;
      =     "DB900_Estado_Mesas".EstadoVI[#MesaDeCarga].Err_Protusion;
      =     #PararElevador;
      BE;

/////////////////////////////////////////////////////////////////////////////////////
/////////////////////////////////////////////////////////////////////////////////////
/////////////////////////////////////////////////////////////////////////////////////
ErrorEnCarga:NOP   0;  // error en la carga
      SET;
      =     "DB900_Estado_Mesas".EstadoVI[#MesaDeCarga].Err_TOut_Avance_E1_E3;
      =     "DB900_Estado_Mesas".EstadoVI[#MesaDeCarga].Error_Mx;
      =     #PararElevador;
      BE;

/////////////////////////////////////////////////////////////////////////////////////
/////////////////////////////////////////////////////////////////////////////////////
/////////////////////////////////////////////////////////////////////////////////////
ErrorMoverPosicionCarga:SET;
      =     #PararElevador;
      =     "DB900_Estado_Mesas".EstadoVI[#MesaDeCarga].Error_Mx;
      =     "DB900_Estado_Mesas".EstadoVI[#MesaDeCarga].Err_Tout_Sacar;
      =     #PararElevador;
      BE;

/////////////////////////////////////////////////////////////////////////////////////
/////////////////////////////////////////////////////////////////////////////////////
/////////////////////////////////////////////////////////////////////////////////////
ErrorMoverPosicionReposo:SET;
      =     #PararElevador;
      =     "DB900_Estado_Mesas".EstadoVI[#MesaDeCarga].Error_Mx;
      =     "DB900_Estado_Mesas".EstadoVI[#MesaDeCarga].Err_Tout_Recoger;
      =     #PararElevador;
      BE;

/////////////////////////////////////////////////////////////////////////////////////
/////////////////////////////////////////////////////////////////////////////////////
/////////////////////////////////////////////////////////////////////////////////////
ErrorDatosCargada:NOP   0;  // error en la carga
      SET;
      =     "DB900_Estado_Mesas".EstadoVI[#MesaDeCarga].Error_Mx;
      =     "DB900_Estado_Mesas".EstadoVI[#MesaDeCarga].Err_DatosPLC;
      =     #PararElevador;
      BE;



NETWORK
TITLE = FINAL DE LA FUNCION
/////////////////////////////////////////////////////////////////////////////////////
/////////////////////////////////////////////////////////////////////////////////////
/////////////////////////////////////////////////////////////////////////////////////
FinFuncion:BE;


END_FUNCTION_BLOCK
